FUNCTION GetMasterLength : REAL
VAR_INPUT
	currentPair : REFERENCE TO PositionMaterials;
END_VAR
VAR
	topLength : REAL;
	leftLength : REAL;
	rightLength : REAL;
	bottomLength : REAL;
	
	topLeftLength : REAL;
	topRightLength : REAL;
	bottomLeftLength : REAL;
	bottomRightLength : REAL;
END_VAR

topLength := GetMaterialLength(currentPair.top);
leftLength := GetMaterialLength(currentPair.left);
rightLength := GetMaterialLength(currentPair.right);
bottomLength := GetMaterialLength(currentPair.bottom);

topLeftLength := GetMaterialLength(currentPair.topLeft);
topRightLength := GetMaterialLength(currentPair.topRight);
bottomLeftLength := GetMaterialLength(currentPair.bottomLeft);
bottomRightLength := GetMaterialLength(currentPair.bottomRight);

GetMasterLength := MAX(topLength, leftLength, rightLength, bottomLength, topLeftLength, topRightLength, bottomLeftLength, bottomRightLength);

END_FUNCTION

(* stored: Version 1.1.0.1, ProductVersion 3.1.4024.11
   POU GetMasterLength: Id {0dbc5c3d-8234-498e-9047-a9c8ff962688}, SpecialFunc None *)
